Yaskawa INFORM job: KELLY.JBI

/JOB
//NAME KELLY
//POS
///NPOS 26,0,0,0
///TOOL 0
///PULSE
C000=14234,56852,-58524,14543,1306,6240
C001=14234,58387,-58749,14546,1251,6229
C002=13262,59038,-57223,14779,1646,6270
C003=13749,58708,-58026,14663,1437,6251
C004=12300,58950,-57643,15048,1551,6224
C005=12300,58330,-57577,15047,1568,6226
C006=13821,58510,-57820,14640,1490,6264
C007=13734,58695,-58031,14669,1437,6253
C008=13629,58175,-59501,14722,1066,6187
C009=13629,57560,-59418,14721,1087,6191
C010=12252,58580,-58169,15069,1417,6204
C011=11474,58319,-58876,15286,1239,6166
C012=12939,58491,-58653,14891,1289,6204
C013=11831,58152,-59685,15198,1030,6152
C014=12552,57922,-60447,15014,832,6137
C015=12143,57900,-60585,15124,798,6131
C016=11204,58390,-58898,15359,1237,6162
C017=12227,57868,-60722,15102,763,6128
C018=11457,57741,-61341,15307,603,6111
C019=11103,57709,-61454,15401,574,6110
C020=10119,57591,-62232,15659,371,6103
C021=9141,57550,-62723,15913,242,6109
C022=7240,57682,-62174,-885,204,6077
C023=6317,57757,-61666,-643,74,6059
C024=8072,57938,-60735,-1102,-165,6032
C025=10622,58246,-59576,15517,1060,6137
//INST
///DATE 2014/09/21 22:32
///ATTR 0,0,0,0,0,0,0,0,0,0,0,0,0,1,0,0
///FRAME BASE
NOP
*Y
MOVJ C000 VJ=50.00 CONT
PAUSE
MOVJ C001 VJ=6.25 CONT
MOVJ C002 VJ=6.25 CONT
MOVJ C003 VJ=6.25 CONT
MOVJ C004 VJ=6.25 CONT
MOVJ C005 VJ=6.25 CONT
MOVJ C006 VJ=6.25 CONT
MOVJ C007 VJ=6.25 CONT
MOVJ C008 VJ=6.25 CONT
MOVJ C009 VJ=6.25 CONT
MOVJ C010 VJ=6.25 CONT
MOVJ C011 VJ=6.25 CONT
MOVJ C012 VJ=6.25 CONT
MOVJ C013 VJ=6.25 CONT
MOVJ C014 VJ=6.25 CONT
MOVJ C015 VJ=6.25 CONT
MOVJ C016 VJ=6.25 CONT
MOVJ C017 VJ=6.25 CONT
MOVJ C018 VJ=6.25 CONT
MOVJ C019 VJ=6.25 CONT
MOVJ C020 VJ=6.25 CONT
MOVJ C021 VJ=6.25 CONT
MOVJ C022 VJ=50.00 CONT
MOVJ C023 VJ=6.25 CONT
MOVJ C024 VJ=6.25 CONT
MOVJ C025 VJ=6.25 CONT
JUMP *Y
END
